{attribute 'qualified_only'}
{attribute 'strict'}
TYPE E_State :
(
    unknown,
    error,
    warning,
    ok
);
END_TYPE

(* stored: Version 1.1.0.1, ProductVersion 3.1.4022.18
   DUT E_State: Id {8f764333-c274-49db-ad7b-896b41852292} *)
